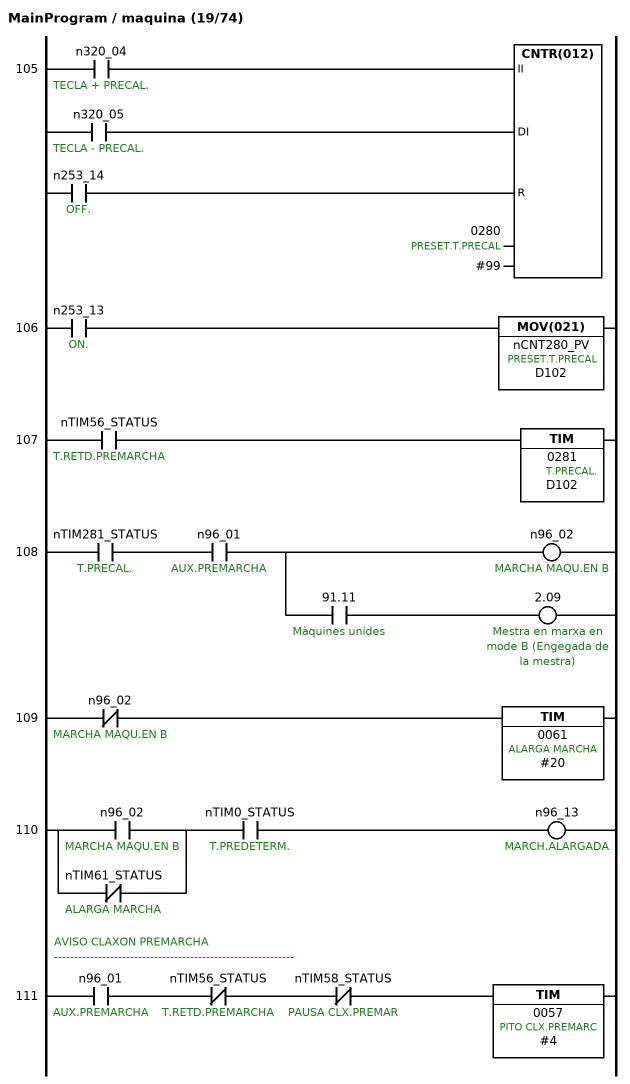
; [picture p24: MainProgram / maquina, rungs 105-111]
; rung 105
LD n320_04  ; TECLA + PRECAL.
LD n320_05  ; TECLA - PRECAL.
LD n253_14  ; OFF.
CNTR(012) 0280 #99  ; PRESET.T.PRECAL
; rung 106
LD n253_13  ; ON.
MOV(021) nCNT280_PV D102  ; PRESET.T.PRECAL
; rung 107
LD nTIM56_STATUS  ; T.RETD.PREMARCHA
TIM 0281 D102  ; T.PRECAL.
; rung 108
LD nTIM281_STATUS  ; T.PRECAL.
AND n96_01  ; AUX.PREMARCHA
OUT n96_02  ; MARCHA MAQU.EN B
AND 91.11  ; Màquines unides
OUT 2.09  ; Mestra en marxa en mode B (Engegada de la mestra)
; rung 109
LDNOT n96_02  ; MARCHA MAQU.EN B
TIM 0061 #20  ; ALARGA MARCHA
; rung 110
LD n96_02  ; MARCHA MAQU.EN B
ORNOT nTIM61_STATUS  ; ALARGA MARCHA
AND nTIM0_STATUS  ; T.PREDETERM.
OUT n96_13  ; MARCH.ALARGADA
; rung 111: AVISO CLAXON PREMARCHA / ------------------------------------------------------------
LD n96_01  ; AUX.PREMARCHA
ANDNOT nTIM56_STATUS  ; T.RETD.PREMARCHA
ANDNOT nTIM58_STATUS  ; PAUSA CLX.PREMAR
TIM 0057 #4  ; PITO CLX.PREMARC

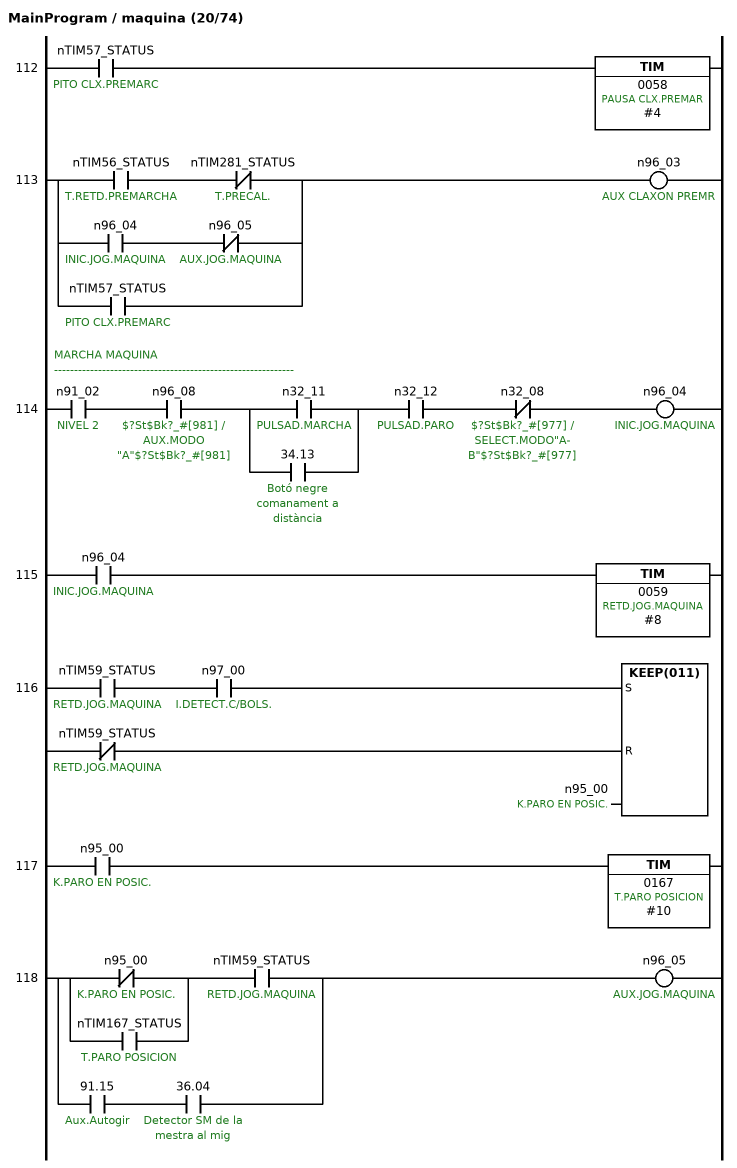
; rung 112
LD nTIM57_STATUS  ; PITO CLX.PREMARC
TIM 0058 #4  ; PAUSA CLX.PREMAR
; rung 113
LD nTIM56_STATUS  ; T.RETD.PREMARCHA
ANDNOT nTIM281_STATUS  ; T.PRECAL.
LD n96_04  ; INIC.JOG.MAQUINA
ANDNOT n96_05  ; AUX.JOG.MAQUINA
ORLD
OR nTIM57_STATUS  ; PITO CLX.PREMARC
OUT n96_03  ; AUX CLAXON PREMR
; rung 114: MARCHA MAQUINA / ------------------------------------------------------------
LD n91_02  ; NIVEL 2
AND n96_08  ; $?St$Bk?_#[981] / AUX.MODO "A"$?St$Bk?_#[981]
LD n32_11  ; PULSAD.MARCHA
OR 34.13  ; Botó negre comanament a distància
ANDLD
AND n32_12  ; PULSAD.PARO
ANDNOT n32_08  ; $?St$Bk?_#[977] / SELECT.MODO"A-B"$?St$Bk?_#[977]
OUT n96_04  ; INIC.JOG.MAQUINA
; rung 115
LD n96_04  ; INIC.JOG.MAQUINA
TIM 0059 #8  ; RETD.JOG.MAQUINA
; rung 116
LD nTIM59_STATUS  ; RETD.JOG.MAQUINA
AND n97_00  ; I.DETECT.C/BOLS.
LDNOT nTIM59_STATUS  ; RETD.JOG.MAQUINA
KEEP(011) n95_00  ; K.PARO EN POSIC.
; rung 117
LD n95_00  ; K.PARO EN POSIC.
TIM 0167 #10  ; T.PARO POSICION
; rung 118
LDNOT n95_00  ; K.PARO EN POSIC.
OR nTIM167_STATUS  ; T.PARO POSICION
AND nTIM59_STATUS  ; RETD.JOG.MAQUINA
LD 91.15  ; Aux.Autogir
AND 36.04  ; Detector SM de la mestra al mig
ORLD
OUT n96_05  ; AUX.JOG.MAQUINA

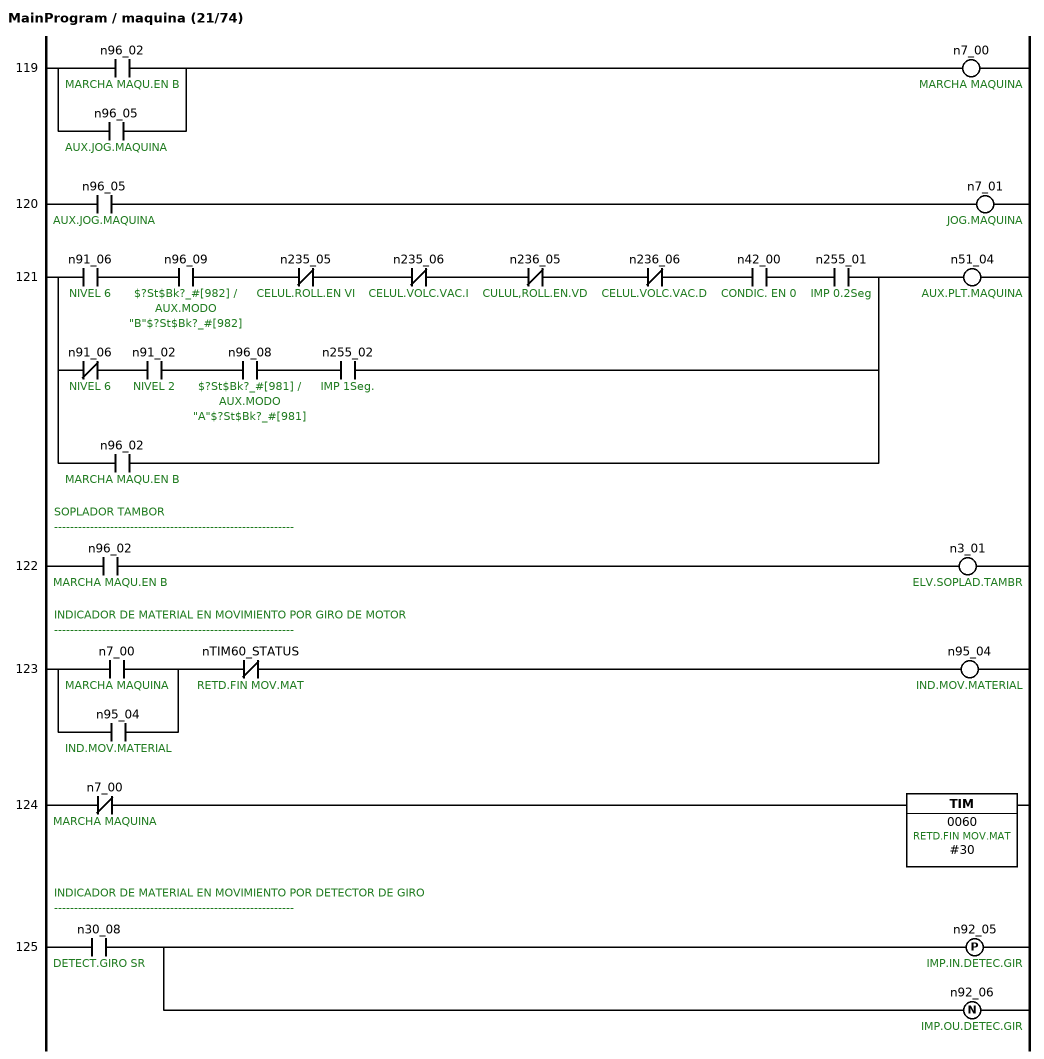
; rung 119
LD n96_02  ; MARCHA MAQU.EN B
OR n96_05  ; AUX.JOG.MAQUINA
OUT n7_00  ; MARCHA MAQUINA
; rung 120
LD n96_05  ; AUX.JOG.MAQUINA
OUT n7_01  ; JOG.MAQUINA
; rung 121
LD n91_06  ; NIVEL 6
AND n96_09  ; $?St$Bk?_#[982] / AUX.MODO "B"$?St$Bk?_#[982]
ANDNOT n235_05  ; CELUL.ROLL.EN VI
ANDNOT n235_06  ; CELUL.VOLC.VAC.I
ANDNOT n236_05  ; CULUL,ROLL.EN.VD
ANDNOT n236_06  ; CELUL.VOLC.VAC.D
AND n42_00  ; CONDIC. EN 0
AND n255_01  ; IMP 0.2Seg
LDNOT n91_06  ; NIVEL 6
AND n91_02  ; NIVEL 2
AND n96_08  ; $?St$Bk?_#[981] / AUX.MODO "A"$?St$Bk?_#[981]
AND n255_02  ; IMP 1Seg.
ORLD
OR n96_02  ; MARCHA MAQU.EN B
OUT n51_04  ; AUX.PLT.MAQUINA
; rung 122: SOPLADOR TAMBOR / ------------------------------------------------------------
LD n96_02  ; MARCHA MAQU.EN B
OUT n3_01  ; ELV.SOPLAD.TAMBR
; rung 123: INDICADOR DE MATERIAL EN MOVIMIENTO POR GIRO DE MOTOR / ------------------------------------------------------------
LD n7_00  ; MARCHA MAQUINA
OR n95_04  ; IND.MOV.MATERIAL
ANDNOT nTIM60_STATUS  ; RETD.FIN MOV.MAT
OUT n95_04  ; IND.MOV.MATERIAL
; rung 124
LDNOT n7_00  ; MARCHA MAQUINA
TIM 0060 #30  ; RETD.FIN MOV.MAT
; rung 125: INDICADOR DE MATERIAL EN MOVIMIENTO POR DETECTOR DE GIRO / ------------------------------------------------------------
LD n30_08  ; DETECT.GIRO SR
DIFU(013) n92_05  ; IMP.IN.DETEC.GIR
DIFD(014) n92_06  ; IMP.OU.DETEC.GIR  // IMPULSO DE SALIDA DETECT.DE GIRO

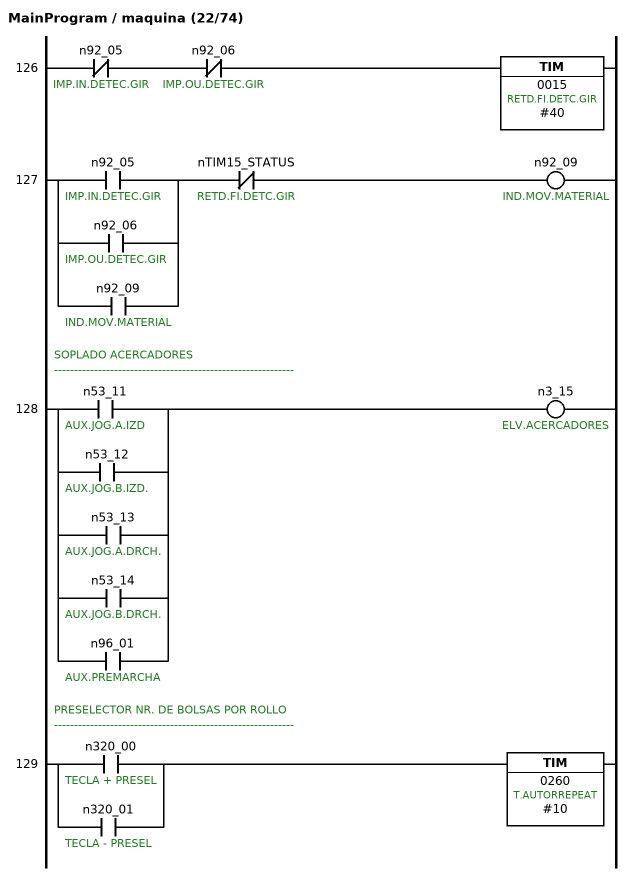
; rung 126
LDNOT n92_05  ; IMP.IN.DETEC.GIR
ANDNOT n92_06  ; IMP.OU.DETEC.GIR
TIM 0015 #40  ; RETD.FI.DETC.GIR  // T.RETARDO FIN DETECTOR DE GIRO
; rung 127
LD n92_05  ; IMP.IN.DETEC.GIR
OR n92_06  ; IMP.OU.DETEC.GIR
OR n92_09  ; IND.MOV.MATERIAL
ANDNOT nTIM15_STATUS  ; RETD.FI.DETC.GIR
OUT n92_09  ; IND.MOV.MATERIAL
; rung 128: SOPLADO ACERCADORES / ------------------------------------------------------------
LD n53_11  ; AUX.JOG.A.IZD
OR n53_12  ; AUX.JOG.B.IZD.
OR n53_13  ; AUX.JOG.A.DRCH.
OR n53_14  ; AUX.JOG.B.DRCH.
OR n96_01  ; AUX.PREMARCHA
OUT n3_15  ; ELV.ACERCADORES
; rung 129: PRESELECTOR NR. DE BOLSAS POR ROLLO / ------------------------------------------------------------
LD n320_00  ; TECLA + PRESEL
OR n320_01  ; TECLA - PRESEL
TIM 0260 #10  ; T.AUTORREPEAT

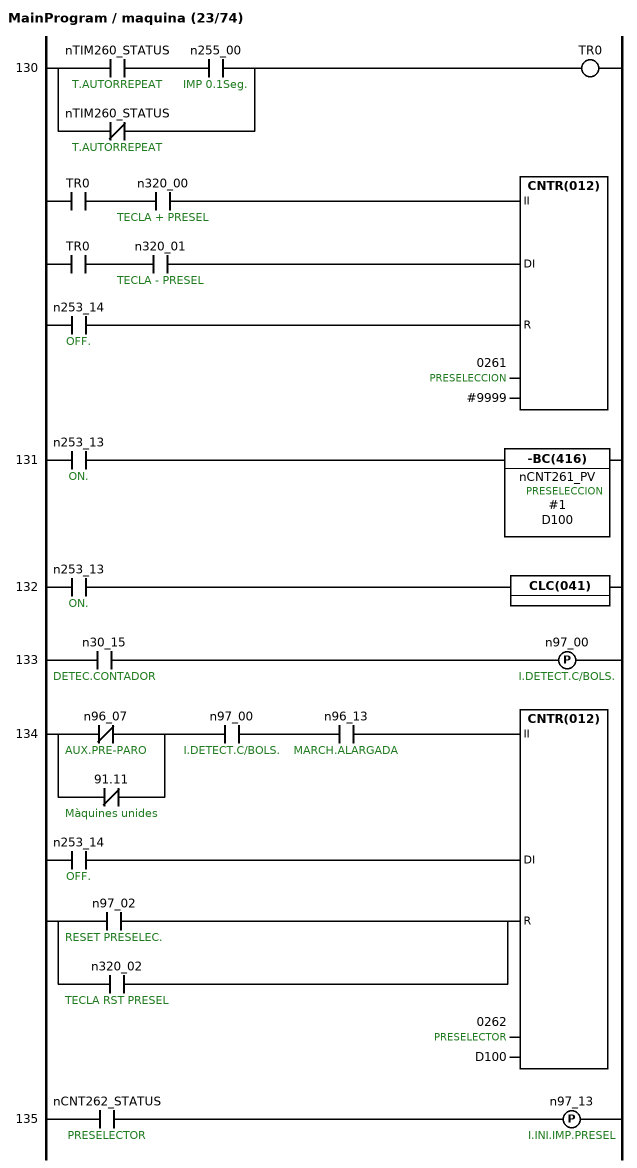
; rung 130
LD nTIM260_STATUS  ; T.AUTORREPEAT
AND n255_00  ; IMP 0.1Seg.
ORNOT nTIM260_STATUS  ; T.AUTORREPEAT
OUT TR0
AND n320_00  ; TECLA + PRESEL
LD TR0
AND n320_01  ; TECLA - PRESEL
LD n253_14  ; OFF.
CNTR(012) 0261 #9999  ; PRESELECCION
; rung 131
LD n253_13  ; ON.
-BC(416) nCNT261_PV #1 D100  ; PRESELECCION
; rung 132
LD n253_13  ; ON.
CLC(041)
; rung 133
LD n30_15  ; DETEC.CONTADOR
DIFU(013) n97_00  ; I.DETECT.C/BOLS.
; rung 134
LDNOT n96_07  ; AUX.PRE-PARO
ORNOT 91.11  ; Màquines unides
AND n97_00  ; I.DETECT.C/BOLS.
AND n96_13  ; MARCH.ALARGADA
LD n253_14  ; OFF.
LD n97_02  ; RESET PRESELEC.
OR n320_02  ; TECLA RST PRESEL
CNTR(012) 0262 D100  ; PRESELECTOR
; rung 135
LD nCNT262_STATUS  ; PRESELECTOR
DIFU(013) n97_13  ; I.INI.IMP.PRESEL

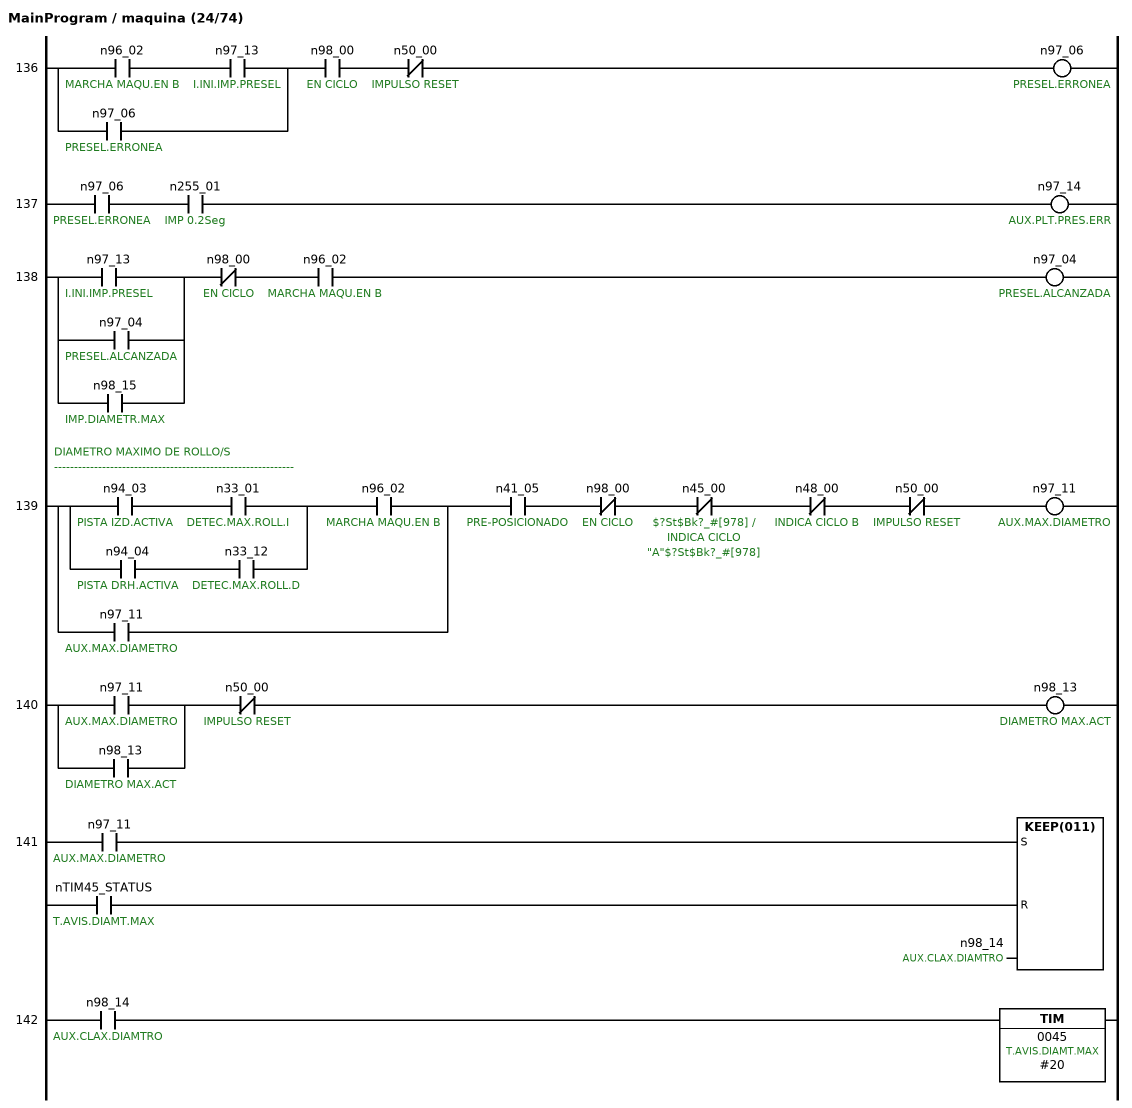
; rung 136
LD n96_02  ; MARCHA MAQU.EN B
AND n97_13  ; I.INI.IMP.PRESEL
OR n97_06  ; PRESEL.ERRONEA
AND n98_00  ; EN CICLO
ANDNOT n50_00  ; IMPULSO RESET
OUT n97_06  ; PRESEL.ERRONEA
; rung 137
LD n97_06  ; PRESEL.ERRONEA
AND n255_01  ; IMP 0.2Seg
OUT n97_14  ; AUX.PLT.PRES.ERR
; rung 138
LD n97_13  ; I.INI.IMP.PRESEL
OR n97_04  ; PRESEL.ALCANZADA
OR n98_15  ; IMP.DIAMETR.MAX
ANDNOT n98_00  ; EN CICLO
AND n96_02  ; MARCHA MAQU.EN B
OUT n97_04  ; PRESEL.ALCANZADA
; rung 139: DIAMETRO MAXIMO DE ROLLO/S / ------------------------------------------------------------
LD n94_03  ; PISTA IZD.ACTIVA
AND n33_01  ; DETEC.MAX.ROLL.I
LD n94_04  ; PISTA DRH.ACTIVA
AND n33_12  ; DETEC.MAX.ROLL.D
ORLD
AND n96_02  ; MARCHA MAQU.EN B
OR n97_11  ; AUX.MAX.DIAMETRO
AND n41_05  ; PRE-POSICIONADO
ANDNOT n98_00  ; EN CICLO
ANDNOT n45_00  ; $?St$Bk?_#[978] / INDICA CICLO "A"$?St$Bk?_#[978]
ANDNOT n48_00  ; INDICA CICLO B
ANDNOT n50_00  ; IMPULSO RESET
OUT n97_11  ; AUX.MAX.DIAMETRO
; rung 140
LD n97_11  ; AUX.MAX.DIAMETRO
OR n98_13  ; DIAMETRO MAX.ACT
ANDNOT n50_00  ; IMPULSO RESET
OUT n98_13  ; DIAMETRO MAX.ACT
; rung 141
LD n97_11  ; AUX.MAX.DIAMETRO
LD nTIM45_STATUS  ; T.AVIS.DIAMT.MAX
KEEP(011) n98_14  ; AUX.CLAX.DIAMTRO
; rung 142
LD n98_14  ; AUX.CLAX.DIAMTRO
TIM 0045 #20  ; T.AVIS.DIAMT.MAX

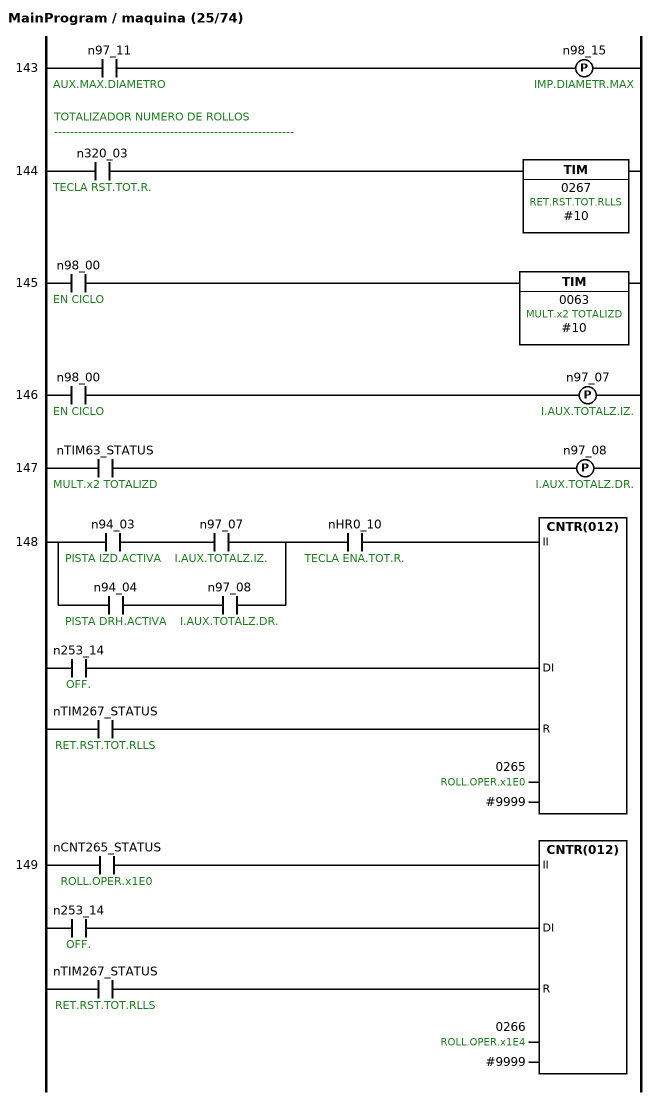
; rung 143
LD n97_11  ; AUX.MAX.DIAMETRO
DIFU(013) n98_15  ; IMP.DIAMETR.MAX
; rung 144: TOTALIZADOR NUMERO DE ROLLOS / ------------------------------------------------------------
LD n320_03  ; TECLA RST.TOT.R.
TIM 0267 #10  ; RET.RST.TOT.RLLS
; rung 145
LD n98_00  ; EN CICLO
TIM 0063 #10  ; MULT.x2 TOTALIZD
; rung 146
LD n98_00  ; EN CICLO
DIFU(013) n97_07  ; I.AUX.TOTALZ.IZ.
; rung 147
LD nTIM63_STATUS  ; MULT.x2 TOTALIZD
DIFU(013) n97_08  ; I.AUX.TOTALZ.DR.
; rung 148
LD n94_03  ; PISTA IZD.ACTIVA
AND n97_07  ; I.AUX.TOTALZ.IZ.
LD n94_04  ; PISTA DRH.ACTIVA
AND n97_08  ; I.AUX.TOTALZ.DR.
ORLD
AND nHR0_10  ; TECLA ENA.TOT.R.
LD n253_14  ; OFF.
LD nTIM267_STATUS  ; RET.RST.TOT.RLLS
CNTR(012) 0265 #9999  ; ROLL.OPER.x1E0
; rung 149
LD nCNT265_STATUS  ; ROLL.OPER.x1E0
LD n253_14  ; OFF.
LD nTIM267_STATUS  ; RET.RST.TOT.RLLS
CNTR(012) 0266 #9999  ; ROLL.OPER.x1E4

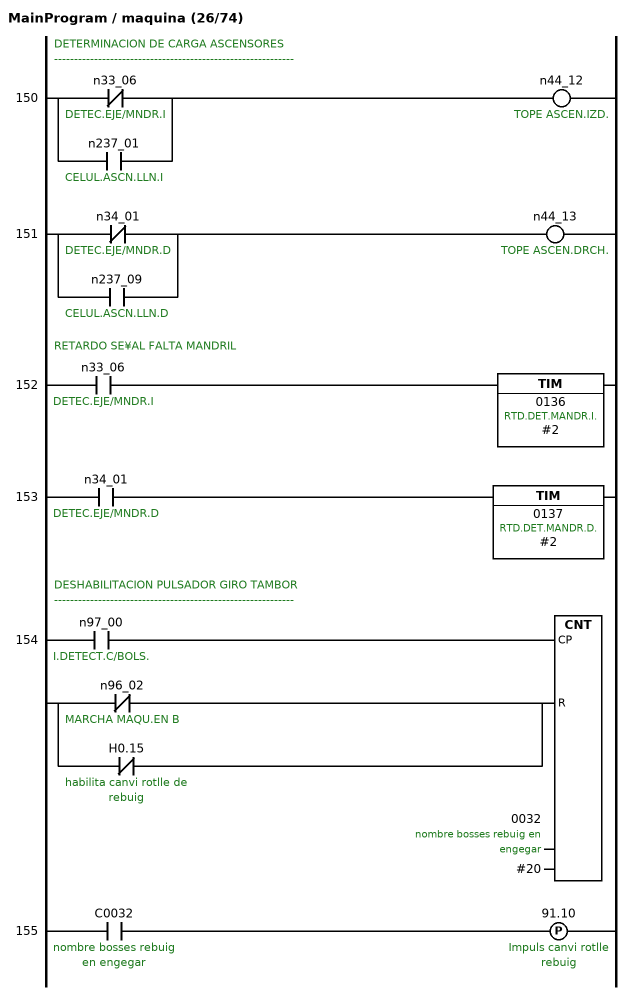
; rung 150: DETERMINACION DE CARGA ASCENSORES / ------------------------------------------------------------
LDNOT n33_06  ; DETEC.EJE/MNDR.I
OR n237_01  ; CELUL.ASCN.LLN.I
OUT n44_12  ; TOPE ASCEN.IZD.
; rung 151
LDNOT n34_01  ; DETEC.EJE/MNDR.D
OR n237_09  ; CELUL.ASCN.LLN.D
OUT n44_13  ; TOPE ASCEN.DRCH.
; rung 152: RETARDO SE¥AL FALTA MANDRIL
LD n33_06  ; DETEC.EJE/MNDR.I
TIM 0136 #2  ; RTD.DET.MANDR.I.
; rung 153
LD n34_01  ; DETEC.EJE/MNDR.D
TIM 0137 #2  ; RTD.DET.MANDR.D.
; rung 154: DESHABILITACION PULSADOR GIRO TAMBOR / ------------------------------------------------------------
LD n97_00  ; I.DETECT.C/BOLS.
LDNOT n96_02  ; MARCHA MAQU.EN B
ORNOT H0.15  ; habilita canvi rotlle de rebuig
CNT 0032 #20  ; nombre bosses rebuig en engegar
; rung 155
LD C0032  ; nombre bosses rebuig en engegar
DIFU(013) 91.10  ; Impuls canvi rotlle rebuig

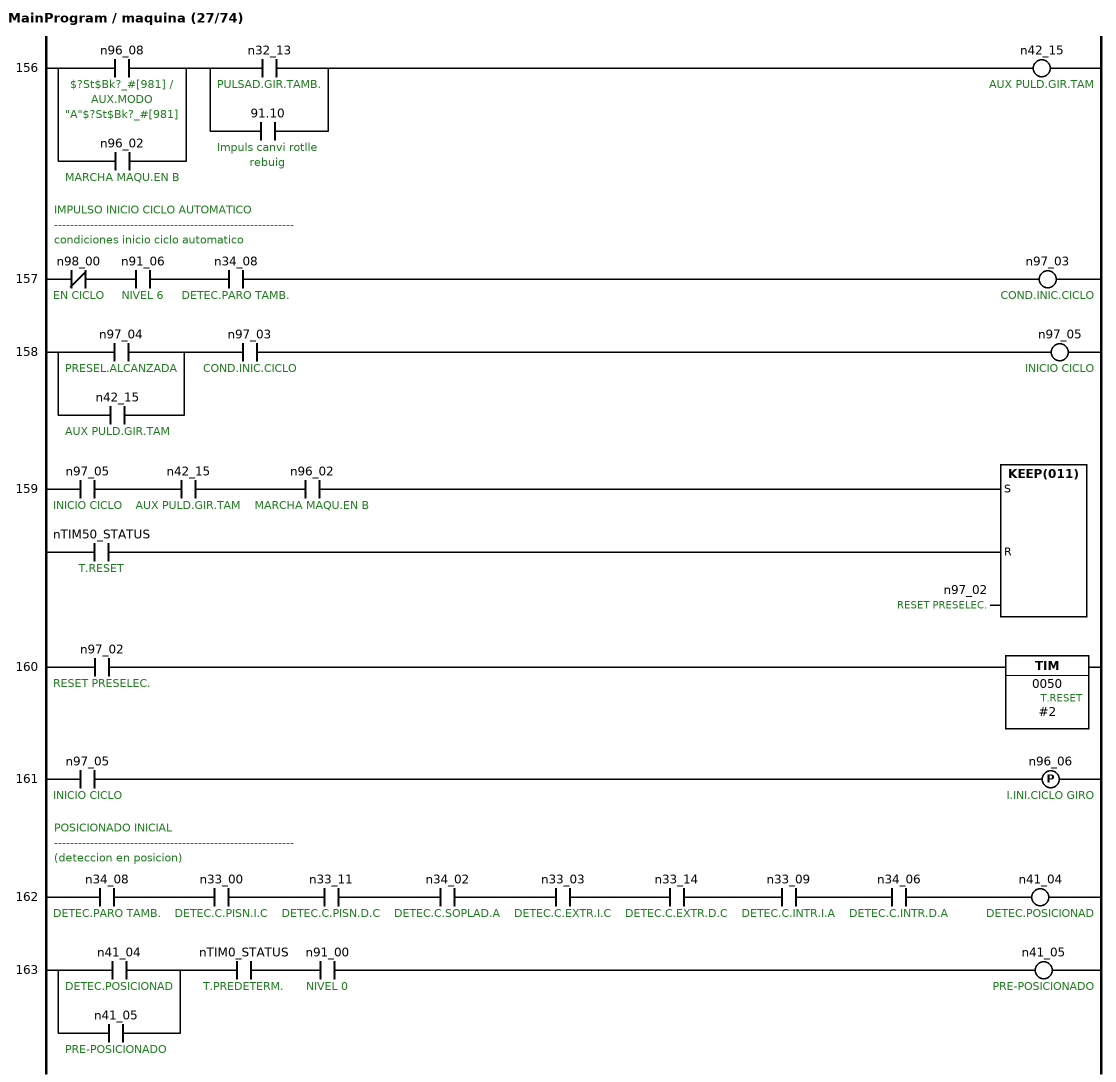
; rung 156
LD n96_08  ; $?St$Bk?_#[981] / AUX.MODO "A"$?St$Bk?_#[981]
OR n96_02  ; MARCHA MAQU.EN B
LD n32_13  ; PULSAD.GIR.TAMB.
OR 91.10  ; Impuls canvi rotlle rebuig
ANDLD
OUT n42_15  ; AUX PULD.GIR.TAM
; rung 157: IMPULSO INICIO CICLO AUTOMATICO / ------------------------------------------------------------ / condiciones inicio ciclo automatico
LDNOT n98_00  ; EN CICLO
AND n91_06  ; NIVEL 6
AND n34_08  ; DETEC.PARO TAMB.
OUT n97_03  ; COND.INIC.CICLO
; rung 158
LD n97_04  ; PRESEL.ALCANZADA
OR n42_15  ; AUX PULD.GIR.TAM
AND n97_03  ; COND.INIC.CICLO
OUT n97_05  ; INICIO CICLO
; rung 159
LD n97_05  ; INICIO CICLO
AND n42_15  ; AUX PULD.GIR.TAM
AND n96_02  ; MARCHA MAQU.EN B
LD nTIM50_STATUS  ; T.RESET
KEEP(011) n97_02  ; RESET PRESELEC.
; rung 160
LD n97_02  ; RESET PRESELEC.
TIM 0050 #2  ; T.RESET
; rung 161
LD n97_05  ; INICIO CICLO
DIFU(013) n96_06  ; I.INI.CICLO GIRO
; rung 162: POSICIONADO INICIAL / ------------------------------------------------------------ / (deteccion en posicion)
LD n34_08  ; DETEC.PARO TAMB.
AND n33_00  ; DETEC.C.PISN.I.C
AND n33_11  ; DETEC.C.PISN.D.C
AND n34_02  ; DETEC.C.SOPLAD.A
AND n33_03  ; DETEC.C.EXTR.I.C
AND n33_14  ; DETEC.C.EXTR.D.C
AND n33_09  ; DETEC.C.INTR.I.A
AND n34_06  ; DETEC.C.INTR.D.A
OUT n41_04  ; DETEC.POSICIONAD
; rung 163
LD n41_04  ; DETEC.POSICIONAD
OR n41_05  ; PRE-POSICIONADO
AND nTIM0_STATUS  ; T.PREDETERM.
AND n91_00  ; NIVEL 0
OUT n41_05  ; PRE-POSICIONADO

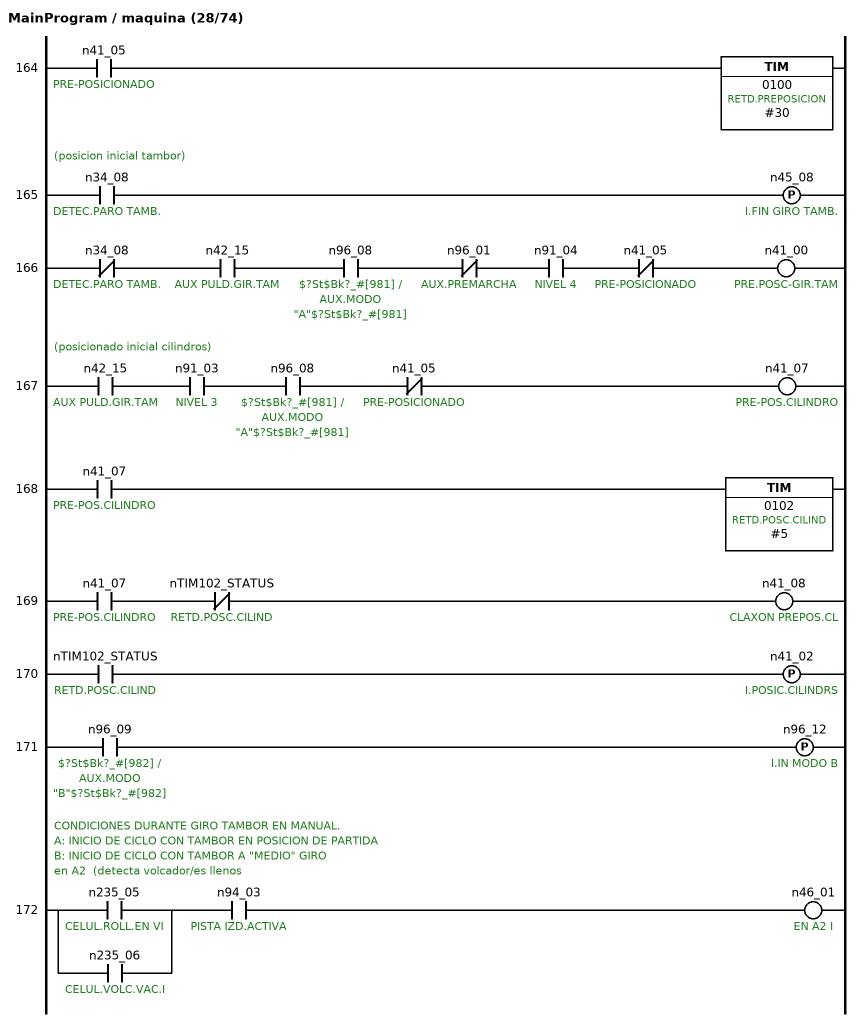
; rung 164
LD n41_05  ; PRE-POSICIONADO
TIM 0100 #30  ; RETD.PREPOSICION
; rung 165: (posicion inicial tambor)
LD n34_08  ; DETEC.PARO TAMB.
DIFU(013) n45_08  ; I.FIN GIRO TAMB.
; rung 166
LDNOT n34_08  ; DETEC.PARO TAMB.
AND n42_15  ; AUX PULD.GIR.TAM
AND n96_08  ; $?St$Bk?_#[981] / AUX.MODO "A"$?St$Bk?_#[981]
ANDNOT n96_01  ; AUX.PREMARCHA
AND n91_04  ; NIVEL 4
ANDNOT n41_05  ; PRE-POSICIONADO
OUT n41_00  ; PRE.POSC-GIR.TAM
; rung 167: (posicionado inicial cilindros)
LD n42_15  ; AUX PULD.GIR.TAM
AND n91_03  ; NIVEL 3
AND n96_08  ; $?St$Bk?_#[981] / AUX.MODO "A"$?St$Bk?_#[981]
ANDNOT n41_05  ; PRE-POSICIONADO
OUT n41_07  ; PRE-POS.CILINDRO
; rung 168
LD n41_07  ; PRE-POS.CILINDRO
TIM 0102 #5  ; RETD.POSC.CILIND
; rung 169
LD n41_07  ; PRE-POS.CILINDRO
ANDNOT nTIM102_STATUS  ; RETD.POSC.CILIND
OUT n41_08  ; CLAXON PREPOS.CL
; rung 170
LD nTIM102_STATUS  ; RETD.POSC.CILIND
DIFU(013) n41_02  ; I.POSIC.CILINDRS
; rung 171
LD n96_09  ; $?St$Bk?_#[982] / AUX.MODO "B"$?St$Bk?_#[982]
DIFU(013) n96_12  ; I.IN MODO B
; rung 172: CONDICIONES DURANTE GIRO TAMBOR EN MANUAL. / A: INICIO DE CICLO CON TAMBOR EN POSICION DE PARTIDA / B: INICIO DE CICLO CON TAMBOR A "MEDIO" GIRO / en A2  (detecta volcador/es llenos
LD n235_05  ; CELUL.ROLL.EN VI
OR n235_06  ; CELUL.VOLC.VAC.I
AND n94_03  ; PISTA IZD.ACTIVA
OUT n46_01  ; EN A2 I

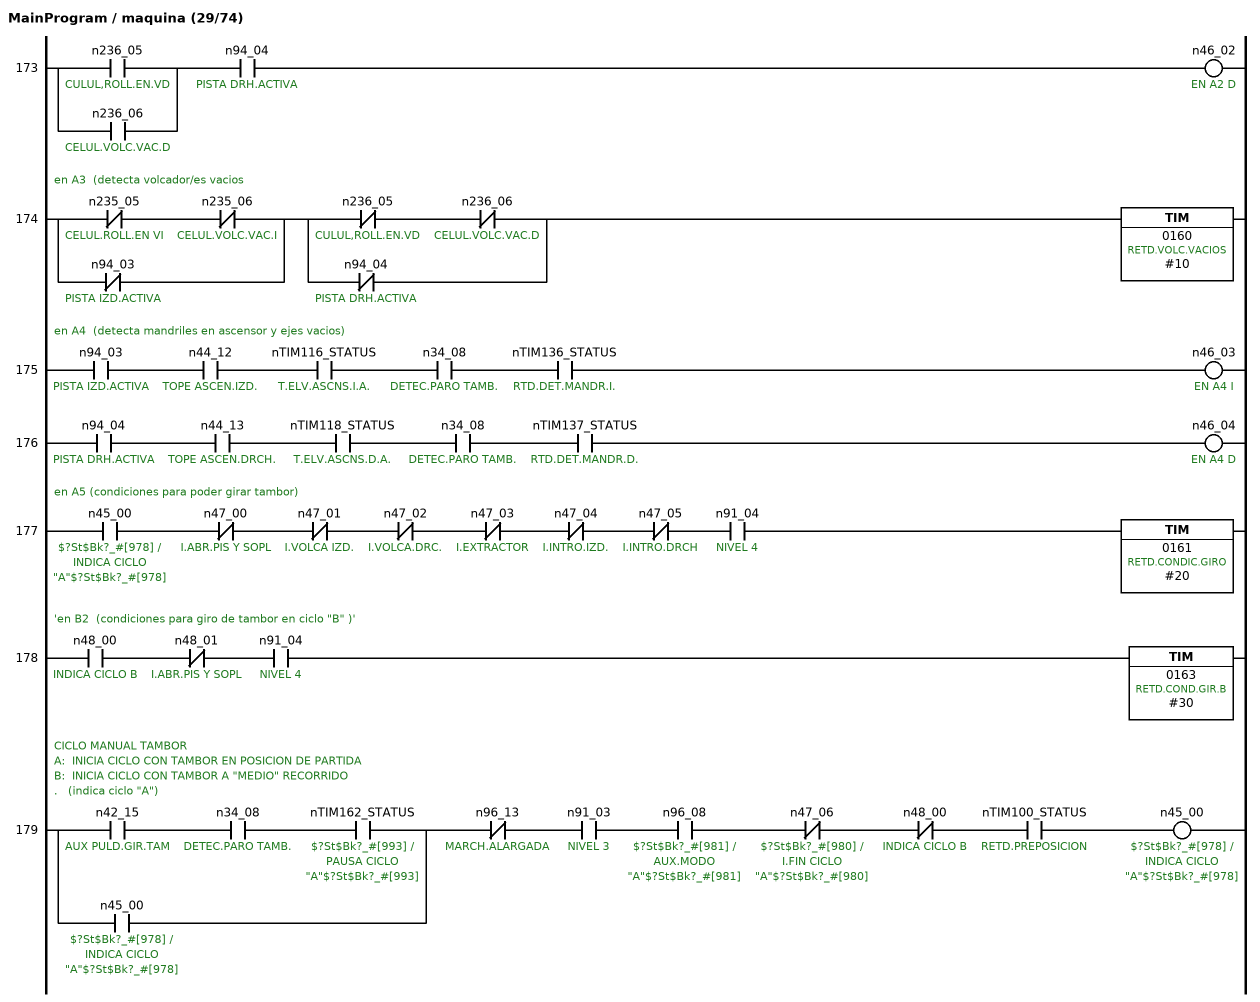
; rung 173
LD n236_05  ; CULUL,ROLL.EN.VD
OR n236_06  ; CELUL.VOLC.VAC.D
AND n94_04  ; PISTA DRH.ACTIVA
OUT n46_02  ; EN A2 D
; rung 174: en A3  (detecta volcador/es vacios
LDNOT n235_05  ; CELUL.ROLL.EN VI
ANDNOT n235_06  ; CELUL.VOLC.VAC.I
ORNOT n94_03  ; PISTA IZD.ACTIVA
LDNOT n236_05  ; CULUL,ROLL.EN.VD
ANDNOT n236_06  ; CELUL.VOLC.VAC.D
ORNOT n94_04  ; PISTA DRH.ACTIVA
ANDLD
TIM 0160 #10  ; RETD.VOLC.VACIOS
; rung 175: en A4  (detecta mandriles en ascensor y ejes vacios)
LD n94_03  ; PISTA IZD.ACTIVA
AND n44_12  ; TOPE ASCEN.IZD.
AND nTIM116_STATUS  ; T.ELV.ASCNS.I.A.
AND n34_08  ; DETEC.PARO TAMB.
AND nTIM136_STATUS  ; RTD.DET.MANDR.I.
OUT n46_03  ; EN A4 I
; rung 176
LD n94_04  ; PISTA DRH.ACTIVA
AND n44_13  ; TOPE ASCEN.DRCH.
AND nTIM118_STATUS  ; T.ELV.ASCNS.D.A.
AND n34_08  ; DETEC.PARO TAMB.
AND nTIM137_STATUS  ; RTD.DET.MANDR.D.
OUT n46_04  ; EN A4 D
; rung 177: en A5 (condiciones para poder girar tambor)
LD n45_00  ; $?St$Bk?_#[978] / INDICA CICLO "A"$?St$Bk?_#[978]
ANDNOT n47_00  ; I.ABR.PIS Y SOPL
ANDNOT n47_01  ; I.VOLCA IZD.
ANDNOT n47_02  ; I.VOLCA.DRC.
ANDNOT n47_03  ; I.EXTRACTOR
ANDNOT n47_04  ; I.INTRO.IZD.
ANDNOT n47_05  ; I.INTRO.DRCH
AND n91_04  ; NIVEL 4
TIM 0161 #20  ; RETD.CONDIC.GIRO
; rung 178: 'en B2  (condiciones para giro de tambor en ciclo "B" )'
LD n48_00  ; INDICA CICLO B
ANDNOT n48_01  ; I.ABR.PIS Y SOPL
AND n91_04  ; NIVEL 4
TIM 0163 #30  ; RETD.COND.GIR.B
; rung 179: CICLO MANUAL TAMBOR / A:  INICIA CICLO CON TAMBOR EN POSICION DE PARTIDA / B:  INICIA CICLO CON TAMBOR A "MEDIO" RECORRIDO / .   (indica ciclo "A")
LD n42_15  ; AUX PULD.GIR.TAM
AND n34_08  ; DETEC.PARO TAMB.
AND nTIM162_STATUS  ; $?St$Bk?_#[993] / PAUSA CICLO "A"$?St$Bk?_#[993]
OR n45_00  ; $?St$Bk?_#[978] / INDICA CICLO "A"$?St$Bk?_#[978]
ANDNOT n96_13  ; MARCH.ALARGADA
AND n91_03  ; NIVEL 3
AND n96_08  ; $?St$Bk?_#[981] / AUX.MODO "A"$?St$Bk?_#[981]
ANDNOT n47_06  ; $?St$Bk?_#[980] / I.FIN CICLO "A"$?St$Bk?_#[980]
ANDNOT n48_00  ; INDICA CICLO B
AND nTIM100_STATUS  ; RETD.PREPOSICION
OUT n45_00  ; $?St$Bk?_#[978] / INDICA CICLO "A"$?St$Bk?_#[978]

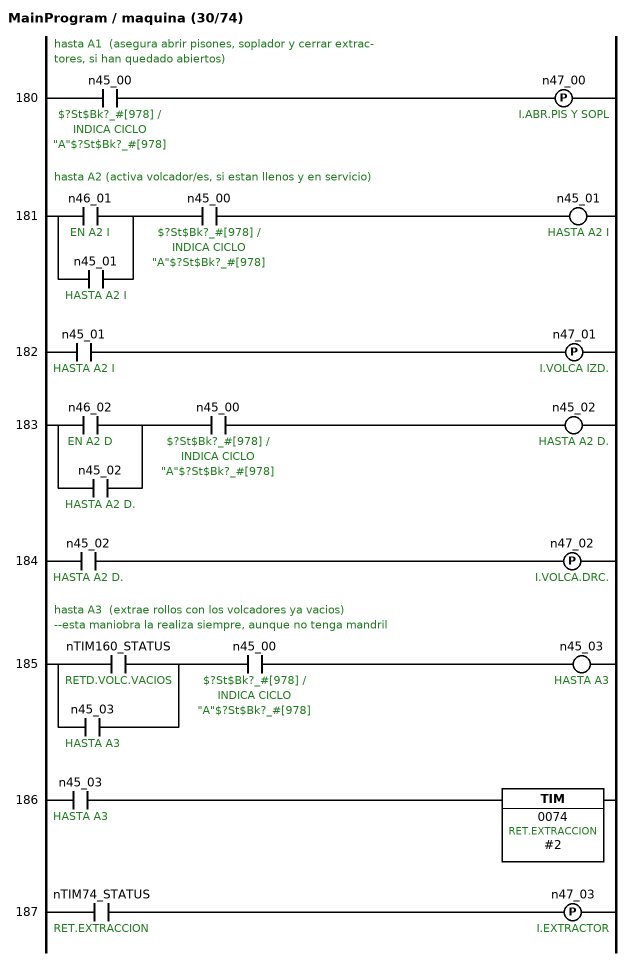
; rung 180: hasta A1  (asegura abrir pisones, soplador y cerrar extrac- / tores, si han quedado abiertos)
LD n45_00  ; $?St$Bk?_#[978] / INDICA CICLO "A"$?St$Bk?_#[978]
DIFU(013) n47_00  ; I.ABR.PIS Y SOPL
; rung 181: hasta A2 (activa volcador/es, si estan llenos y en servicio)
LD n46_01  ; EN A2 I
OR n45_01  ; HASTA A2 I
AND n45_00  ; $?St$Bk?_#[978] / INDICA CICLO "A"$?St$Bk?_#[978]
OUT n45_01  ; HASTA A2 I
; rung 182
LD n45_01  ; HASTA A2 I
DIFU(013) n47_01  ; I.VOLCA IZD.
; rung 183
LD n46_02  ; EN A2 D
OR n45_02  ; HASTA A2 D.
AND n45_00  ; $?St$Bk?_#[978] / INDICA CICLO "A"$?St$Bk?_#[978]
OUT n45_02  ; HASTA A2 D.
; rung 184
LD n45_02  ; HASTA A2 D.
DIFU(013) n47_02  ; I.VOLCA.DRC.
; rung 185: hasta A3  (extrae rollos con los volcadores ya vacios) / --esta maniobra la realiza siempre, aunque no tenga mandril
LD nTIM160_STATUS  ; RETD.VOLC.VACIOS
OR n45_03  ; HASTA A3
AND n45_00  ; $?St$Bk?_#[978] / INDICA CICLO "A"$?St$Bk?_#[978]
OUT n45_03  ; HASTA A3
; rung 186
LD n45_03  ; HASTA A3
TIM 0074 #2  ; RET.EXTRACCION
; rung 187
LD nTIM74_STATUS  ; RET.EXTRACCION
DIFU(013) n47_03  ; I.EXTRACTOR

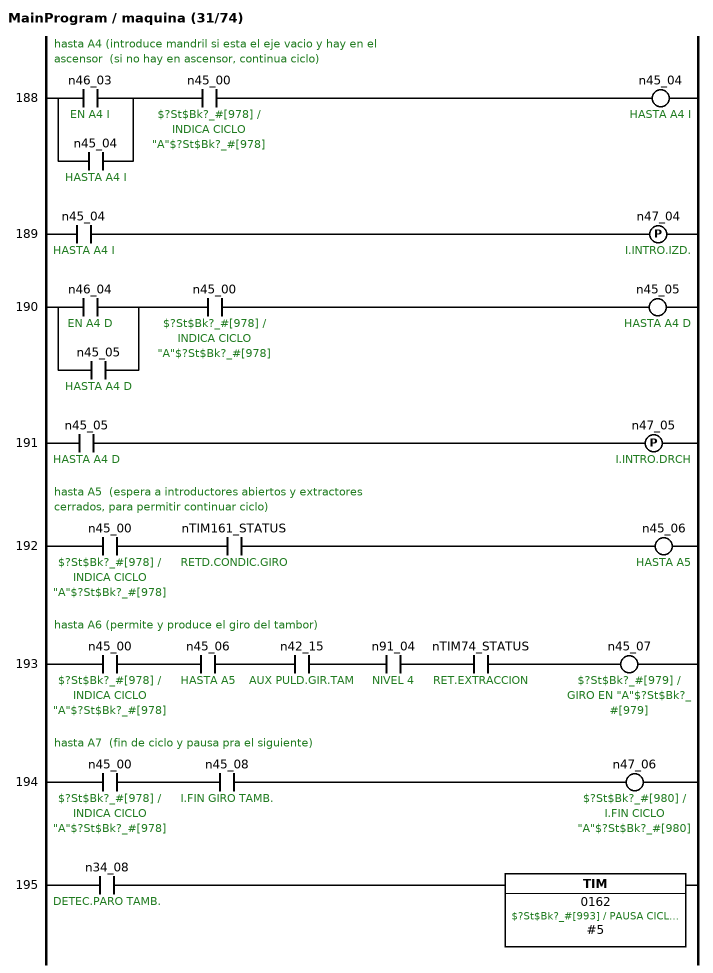
; rung 188: hasta A4 (introduce mandril si esta el eje vacio y hay en el / ascensor  (si no hay en ascensor, continua ciclo)
LD n46_03  ; EN A4 I
OR n45_04  ; HASTA A4 I
AND n45_00  ; $?St$Bk?_#[978] / INDICA CICLO "A"$?St$Bk?_#[978]
OUT n45_04  ; HASTA A4 I
; rung 189
LD n45_04  ; HASTA A4 I
DIFU(013) n47_04  ; I.INTRO.IZD.
; rung 190
LD n46_04  ; EN A4 D
OR n45_05  ; HASTA A4 D
AND n45_00  ; $?St$Bk?_#[978] / INDICA CICLO "A"$?St$Bk?_#[978]
OUT n45_05  ; HASTA A4 D
; rung 191
LD n45_05  ; HASTA A4 D
DIFU(013) n47_05  ; I.INTRO.DRCH
; rung 192: hasta A5  (espera a introductores abiertos y extractores / cerrados, para permitir continuar ciclo)
LD n45_00  ; $?St$Bk?_#[978] / INDICA CICLO "A"$?St$Bk?_#[978]
AND nTIM161_STATUS  ; RETD.CONDIC.GIRO
OUT n45_06  ; HASTA A5
; rung 193: hasta A6 (permite y produce el giro del tambor)
LD n45_00  ; $?St$Bk?_#[978] / INDICA CICLO "A"$?St$Bk?_#[978]
AND n45_06  ; HASTA A5
AND n42_15  ; AUX PULD.GIR.TAM
AND n91_04  ; NIVEL 4
AND nTIM74_STATUS  ; RET.EXTRACCION
OUT n45_07  ; $?St$Bk?_#[979] / GIRO EN "A"$?St$Bk?_#[979]
; rung 194: hasta A7  (fin de ciclo y pausa pra el siguiente)
LD n45_00  ; $?St$Bk?_#[978] / INDICA CICLO "A"$?St$Bk?_#[978]
AND n45_08  ; I.FIN GIRO TAMB.
OUT n47_06  ; $?St$Bk?_#[980] / I.FIN CICLO "A"$?St$Bk?_#[980]
; rung 195
LD n34_08  ; DETEC.PARO TAMB.
TIM 0162 #5  ; $?St$Bk?_#[993] / PAUSA CICLO "A"$?St$Bk?_#[993]

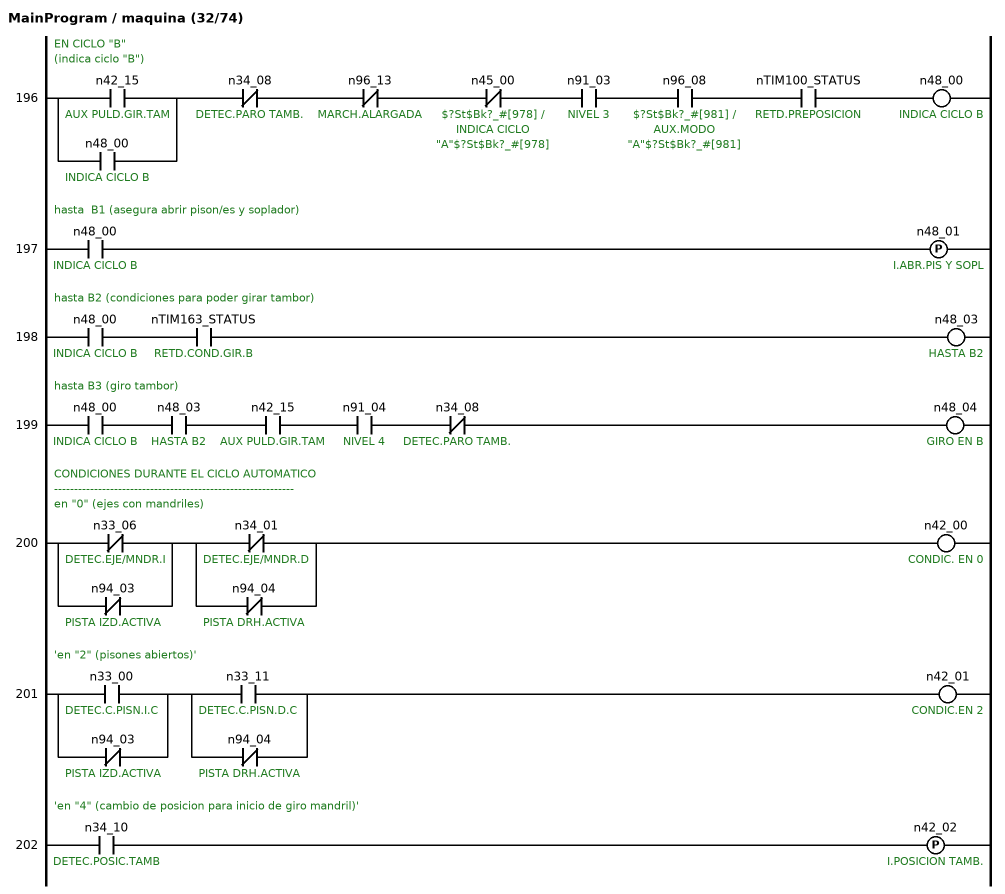
; rung 196: EN CICLO "B" / (indica ciclo "B")
LD n42_15  ; AUX PULD.GIR.TAM
OR n48_00  ; INDICA CICLO B
ANDNOT n34_08  ; DETEC.PARO TAMB.
ANDNOT n96_13  ; MARCH.ALARGADA
ANDNOT n45_00  ; $?St$Bk?_#[978] / INDICA CICLO "A"$?St$Bk?_#[978]
AND n91_03  ; NIVEL 3
AND n96_08  ; $?St$Bk?_#[981] / AUX.MODO "A"$?St$Bk?_#[981]
AND nTIM100_STATUS  ; RETD.PREPOSICION
OUT n48_00  ; INDICA CICLO B
; rung 197: hasta  B1 (asegura abrir pison/es y soplador)
LD n48_00  ; INDICA CICLO B
DIFU(013) n48_01  ; I.ABR.PIS Y SOPL
; rung 198: hasta B2 (condiciones para poder girar tambor)
LD n48_00  ; INDICA CICLO B
AND nTIM163_STATUS  ; RETD.COND.GIR.B
OUT n48_03  ; HASTA B2
; rung 199: hasta B3 (giro tambor)
LD n48_00  ; INDICA CICLO B
AND n48_03  ; HASTA B2
AND n42_15  ; AUX PULD.GIR.TAM
AND n91_04  ; NIVEL 4
ANDNOT n34_08  ; DETEC.PARO TAMB.
OUT n48_04  ; GIRO EN B
; rung 200: CONDICIONES DURANTE EL CICLO AUTOMATICO / ------------------------------------------------------------ / en "0" (ejes con mandriles)
LDNOT n33_06  ; DETEC.EJE/MNDR.I
ORNOT n94_03  ; PISTA IZD.ACTIVA
LDNOT n34_01  ; DETEC.EJE/MNDR.D
ORNOT n94_04  ; PISTA DRH.ACTIVA
ANDLD
OUT n42_00  ; CONDIC. EN 0
; rung 201: 'en "2" (pisones abiertos)'
LD n33_00  ; DETEC.C.PISN.I.C
ORNOT n94_03  ; PISTA IZD.ACTIVA
LD n33_11  ; DETEC.C.PISN.D.C
ORNOT n94_04  ; PISTA DRH.ACTIVA
ANDLD
OUT n42_01  ; CONDIC.EN 2
; rung 202: 'en "4" (cambio de posicion para inicio de giro mandril)'
LD n34_10  ; DETEC.POSIC.TAMB
DIFU(013) n42_02  ; I.POSICION TAMB.

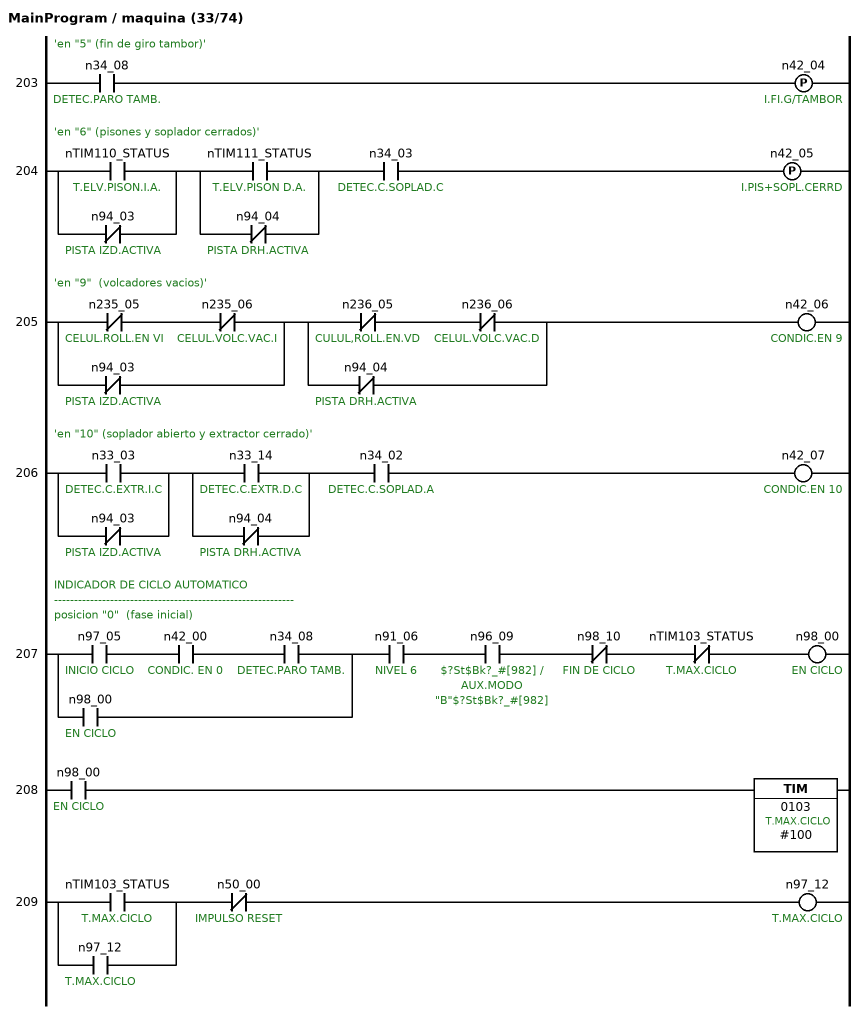
; rung 203: 'en "5" (fin de giro tambor)'
LD n34_08  ; DETEC.PARO TAMB.
DIFU(013) n42_04  ; I.FI.G/TAMBOR
; rung 204: 'en "6" (pisones y soplador cerrados)'
LD nTIM110_STATUS  ; T.ELV.PISON.I.A.
ORNOT n94_03  ; PISTA IZD.ACTIVA
LD nTIM111_STATUS  ; T.ELV.PISON D.A.
ORNOT n94_04  ; PISTA DRH.ACTIVA
ANDLD
AND n34_03  ; DETEC.C.SOPLAD.C
DIFU(013) n42_05  ; I.PIS+SOPL.CERRD
; rung 205: 'en "9"  (volcadores vacios)'
LDNOT n235_05  ; CELUL.ROLL.EN VI
ANDNOT n235_06  ; CELUL.VOLC.VAC.I
ORNOT n94_03  ; PISTA IZD.ACTIVA
LDNOT n236_05  ; CULUL,ROLL.EN.VD
ANDNOT n236_06  ; CELUL.VOLC.VAC.D
ORNOT n94_04  ; PISTA DRH.ACTIVA
ANDLD
OUT n42_06  ; CONDIC.EN 9
; rung 206: 'en "10" (soplador abierto y extractor cerrado)'
LD n33_03  ; DETEC.C.EXTR.I.C
ORNOT n94_03  ; PISTA IZD.ACTIVA
LD n33_14  ; DETEC.C.EXTR.D.C
ORNOT n94_04  ; PISTA DRH.ACTIVA
ANDLD
AND n34_02  ; DETEC.C.SOPLAD.A
OUT n42_07  ; CONDIC.EN 10
; rung 207: INDICADOR DE CICLO AUTOMATICO / ------------------------------------------------------------ / posicion "0"  (fase inicial)
LD n97_05  ; INICIO CICLO
AND n42_00  ; CONDIC. EN 0
AND n34_08  ; DETEC.PARO TAMB.
OR n98_00  ; EN CICLO
AND n91_06  ; NIVEL 6
AND n96_09  ; $?St$Bk?_#[982] / AUX.MODO "B"$?St$Bk?_#[982]
ANDNOT n98_10  ; FIN DE CICLO
ANDNOT nTIM103_STATUS  ; T.MAX.CICLO
OUT n98_00  ; EN CICLO
; rung 208
LD n98_00  ; EN CICLO
TIM 0103 #100  ; T.MAX.CICLO
; rung 209
LD nTIM103_STATUS  ; T.MAX.CICLO
OR n97_12  ; T.MAX.CICLO
ANDNOT n50_00  ; IMPULSO RESET
OUT n97_12  ; T.MAX.CICLO

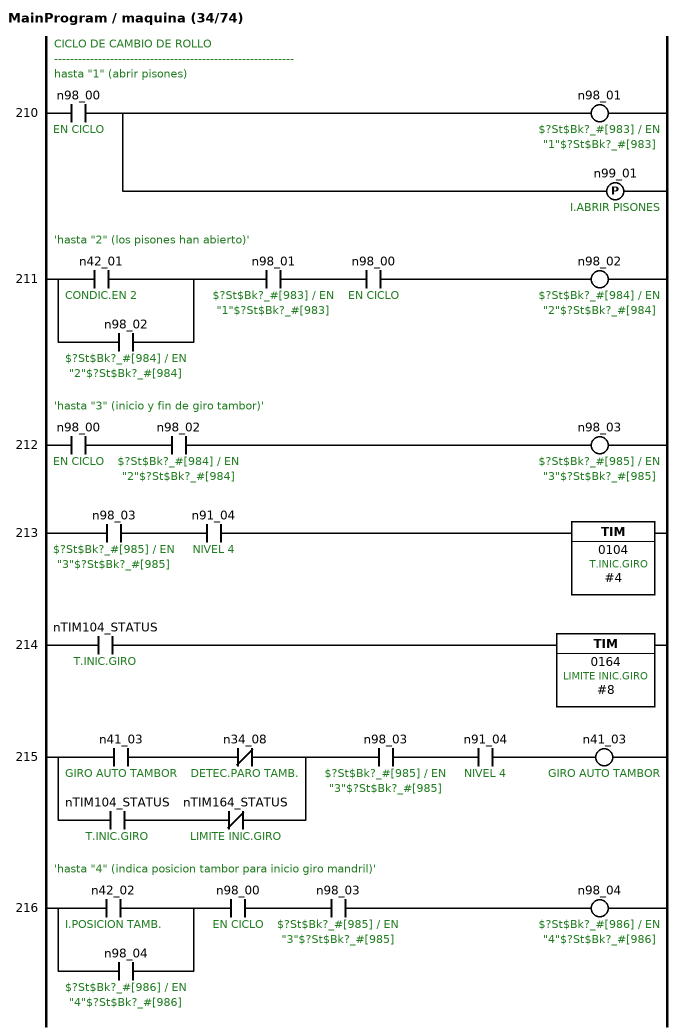
; rung 210: CICLO DE CAMBIO DE ROLLO / ------------------------------------------------------------ / hasta "1" (abrir pisones)
LD n98_00  ; EN CICLO
OUT n98_01  ; $?St$Bk?_#[983] / EN "1"$?St$Bk?_#[983]
DIFU(013) n99_01  ; I.ABRIR PISONES
; rung 211: 'hasta "2" (los pisones han abierto)'
LD n42_01  ; CONDIC.EN 2
OR n98_02  ; $?St$Bk?_#[984] / EN "2"$?St$Bk?_#[984]
AND n98_01  ; $?St$Bk?_#[983] / EN "1"$?St$Bk?_#[983]
AND n98_00  ; EN CICLO
OUT n98_02  ; $?St$Bk?_#[984] / EN "2"$?St$Bk?_#[984]
; rung 212: 'hasta "3" (inicio y fin de giro tambor)'
LD n98_00  ; EN CICLO
AND n98_02  ; $?St$Bk?_#[984] / EN "2"$?St$Bk?_#[984]
OUT n98_03  ; $?St$Bk?_#[985] / EN "3"$?St$Bk?_#[985]
; rung 213
LD n98_03  ; $?St$Bk?_#[985] / EN "3"$?St$Bk?_#[985]
AND n91_04  ; NIVEL 4
TIM 0104 #4  ; T.INIC.GIRO
; rung 214
LD nTIM104_STATUS  ; T.INIC.GIRO
TIM 0164 #8  ; LIMITE INIC.GIRO
; rung 215
LD n41_03  ; GIRO AUTO TAMBOR
ANDNOT n34_08  ; DETEC.PARO TAMB.
LD nTIM104_STATUS  ; T.INIC.GIRO
ANDNOT nTIM164_STATUS  ; LIMITE INIC.GIRO
ORLD
AND n98_03  ; $?St$Bk?_#[985] / EN "3"$?St$Bk?_#[985]
AND n91_04  ; NIVEL 4
OUT n41_03  ; GIRO AUTO TAMBOR
; rung 216: 'hasta "4" (indica posicion tambor para inicio giro mandril)'
LD n42_02  ; I.POSICION TAMB.
OR n98_04  ; $?St$Bk?_#[986] / EN "4"$?St$Bk?_#[986]
AND n98_00  ; EN CICLO
AND n98_03  ; $?St$Bk?_#[985] / EN "3"$?St$Bk?_#[985]
OUT n98_04  ; $?St$Bk?_#[986] / EN "4"$?St$Bk?_#[986]

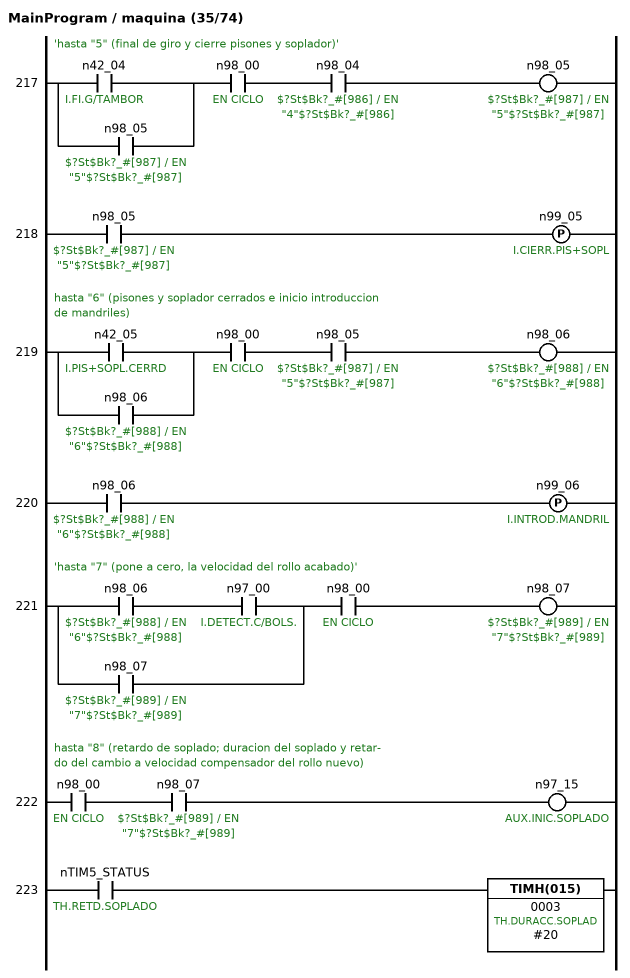
; rung 217: 'hasta "5" (final de giro y cierre pisones y soplador)'
LD n42_04  ; I.FI.G/TAMBOR
OR n98_05  ; $?St$Bk?_#[987] / EN "5"$?St$Bk?_#[987]
AND n98_00  ; EN CICLO
AND n98_04  ; $?St$Bk?_#[986] / EN "4"$?St$Bk?_#[986]
OUT n98_05  ; $?St$Bk?_#[987] / EN "5"$?St$Bk?_#[987]
; rung 218
LD n98_05  ; $?St$Bk?_#[987] / EN "5"$?St$Bk?_#[987]
DIFU(013) n99_05  ; I.CIERR.PIS+SOPL
; rung 219: hasta "6" (pisones y soplador cerrados e inicio introduccion / de mandriles)
LD n42_05  ; I.PIS+SOPL.CERRD
OR n98_06  ; $?St$Bk?_#[988] / EN "6"$?St$Bk?_#[988]
AND n98_00  ; EN CICLO
AND n98_05  ; $?St$Bk?_#[987] / EN "5"$?St$Bk?_#[987]
OUT n98_06  ; $?St$Bk?_#[988] / EN "6"$?St$Bk?_#[988]
; rung 220
LD n98_06  ; $?St$Bk?_#[988] / EN "6"$?St$Bk?_#[988]
DIFU(013) n99_06  ; I.INTROD.MANDRIL
; rung 221: 'hasta "7" (pone a cero, la velocidad del rollo acabado)'
LD n98_06  ; $?St$Bk?_#[988] / EN "6"$?St$Bk?_#[988]
AND n97_00  ; I.DETECT.C/BOLS.
OR n98_07  ; $?St$Bk?_#[989] / EN "7"$?St$Bk?_#[989]
AND n98_00  ; EN CICLO
OUT n98_07  ; $?St$Bk?_#[989] / EN "7"$?St$Bk?_#[989]
; rung 222: hasta "8" (retardo de soplado; duracion del soplado y retar- / do del cambio a velocidad compensador del rollo nuevo)
LD n98_00  ; EN CICLO
AND n98_07  ; $?St$Bk?_#[989] / EN "7"$?St$Bk?_#[989]
OUT n97_15  ; AUX.INIC.SOPLADO
; rung 223
LD nTIM5_STATUS  ; TH.RETD.SOPLADO
TIMH(015) 0003 #20  ; TH.DURACC.SOPLAD

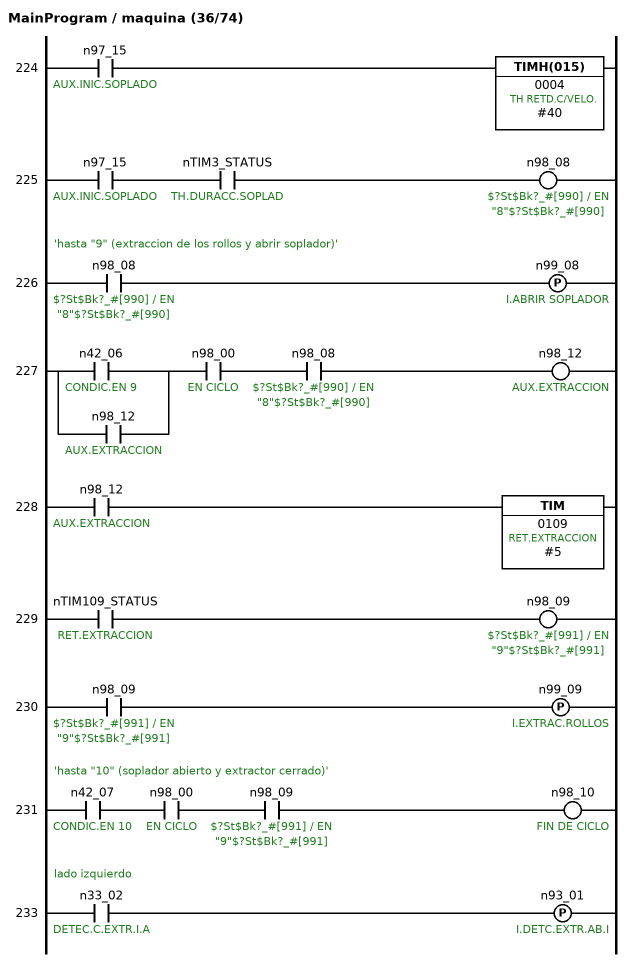
; rung 224
LD n97_15  ; AUX.INIC.SOPLADO
TIMH(015) 0004 #40  ; TH RETD.C/VELO.
; rung 225
LD n97_15  ; AUX.INIC.SOPLADO
AND nTIM3_STATUS  ; TH.DURACC.SOPLAD
OUT n98_08  ; $?St$Bk?_#[990] / EN "8"$?St$Bk?_#[990]
; rung 226: 'hasta "9" (extraccion de los rollos y abrir soplador)'
LD n98_08  ; $?St$Bk?_#[990] / EN "8"$?St$Bk?_#[990]
DIFU(013) n99_08  ; I.ABRIR SOPLADOR
; rung 227
LD n42_06  ; CONDIC.EN 9
OR n98_12  ; AUX.EXTRACCION
AND n98_00  ; EN CICLO
AND n98_08  ; $?St$Bk?_#[990] / EN "8"$?St$Bk?_#[990]
OUT n98_12  ; AUX.EXTRACCION
; rung 228
LD n98_12  ; AUX.EXTRACCION
TIM 0109 #5  ; RET.EXTRACCION
; rung 229
LD nTIM109_STATUS  ; RET.EXTRACCION
OUT n98_09  ; $?St$Bk?_#[991] / EN "9"$?St$Bk?_#[991]
; rung 230
LD n98_09  ; $?St$Bk?_#[991] / EN "9"$?St$Bk?_#[991]
DIFU(013) n99_09  ; I.EXTRAC.ROLLOS
; rung 231: 'hasta "10" (soplador abierto y extractor cerrado)'
LD n42_07  ; CONDIC.EN 10
AND n98_00  ; EN CICLO
AND n98_09  ; $?St$Bk?_#[991] / EN "9"$?St$Bk?_#[991]
OUT n98_10  ; FIN DE CICLO
; rung 232: VIGILANCIA ROLLOS NO CAIDOS DEL EJE REBOBINADOR / ------------------------------------------------------------
; rung 233: lado izquierdo
LD n33_02  ; DETEC.C.EXTR.I.A
DIFU(013) n93_01  ; I.DETC.EXTR.AB.I

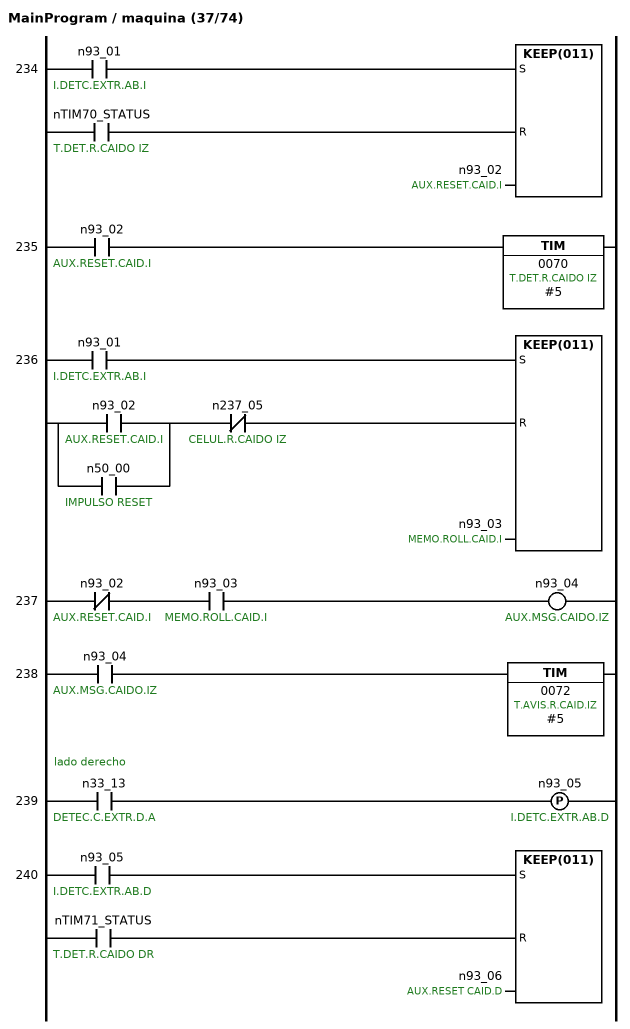
; rung 234
LD n93_01  ; I.DETC.EXTR.AB.I
LD nTIM70_STATUS  ; T.DET.R.CAIDO IZ
KEEP(011) n93_02  ; AUX.RESET.CAID.I
; rung 235
LD n93_02  ; AUX.RESET.CAID.I
TIM 0070 #5  ; T.DET.R.CAIDO IZ
; rung 236
LD n93_01  ; I.DETC.EXTR.AB.I
LD n93_02  ; AUX.RESET.CAID.I
OR n50_00  ; IMPULSO RESET
ANDNOT n237_05  ; CELUL.R.CAIDO IZ
KEEP(011) n93_03  ; MEMO.ROLL.CAID.I
; rung 237
LDNOT n93_02  ; AUX.RESET.CAID.I
AND n93_03  ; MEMO.ROLL.CAID.I
OUT n93_04  ; AUX.MSG.CAIDO.IZ
; rung 238
LD n93_04  ; AUX.MSG.CAIDO.IZ
TIM 0072 #5  ; T.AVIS.R.CAID.IZ
; rung 239: lado derecho
LD n33_13  ; DETEC.C.EXTR.D.A
DIFU(013) n93_05  ; I.DETC.EXTR.AB.D
; rung 240
LD n93_05  ; I.DETC.EXTR.AB.D
LD nTIM71_STATUS  ; T.DET.R.CAIDO DR
KEEP(011) n93_06  ; AUX.RESET CAID.D

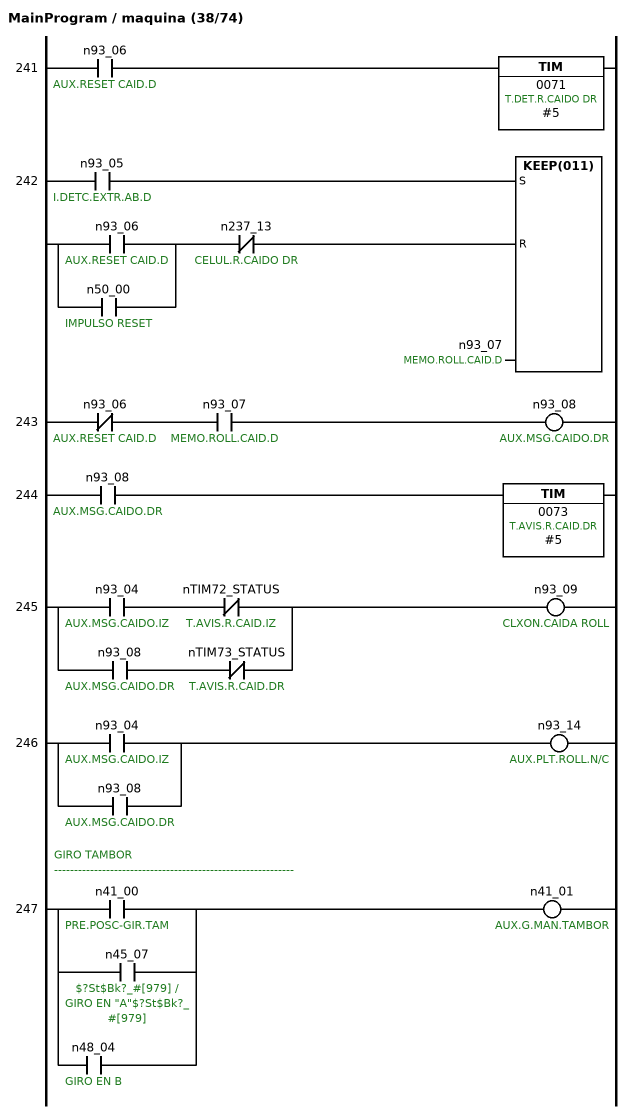
; rung 241
LD n93_06  ; AUX.RESET CAID.D
TIM 0071 #5  ; T.DET.R.CAIDO DR
; rung 242
LD n93_05  ; I.DETC.EXTR.AB.D
LD n93_06  ; AUX.RESET CAID.D
OR n50_00  ; IMPULSO RESET
ANDNOT n237_13  ; CELUL.R.CAIDO DR
KEEP(011) n93_07  ; MEMO.ROLL.CAID.D
; rung 243
LDNOT n93_06  ; AUX.RESET CAID.D
AND n93_07  ; MEMO.ROLL.CAID.D
OUT n93_08  ; AUX.MSG.CAIDO.DR
; rung 244
LD n93_08  ; AUX.MSG.CAIDO.DR
TIM 0073 #5  ; T.AVIS.R.CAID.DR
; rung 245
LD n93_04  ; AUX.MSG.CAIDO.IZ
ANDNOT nTIM72_STATUS  ; T.AVIS.R.CAID.IZ
LD n93_08  ; AUX.MSG.CAIDO.DR
ANDNOT nTIM73_STATUS  ; T.AVIS.R.CAID.DR
ORLD
OUT n93_09  ; CLXON.CAIDA ROLL
; rung 246
LD n93_04  ; AUX.MSG.CAIDO.IZ
OR n93_08  ; AUX.MSG.CAIDO.DR
OUT n93_14  ; AUX.PLT.ROLL.N/C
; rung 247: GIRO TAMBOR / ------------------------------------------------------------
LD n41_00  ; PRE.POSC-GIR.TAM
OR n45_07  ; $?St$Bk?_#[979] / GIRO EN "A"$?St$Bk?_#[979]
OR n48_04  ; GIRO EN B
OUT n41_01  ; AUX.G.MAN.TAMBOR

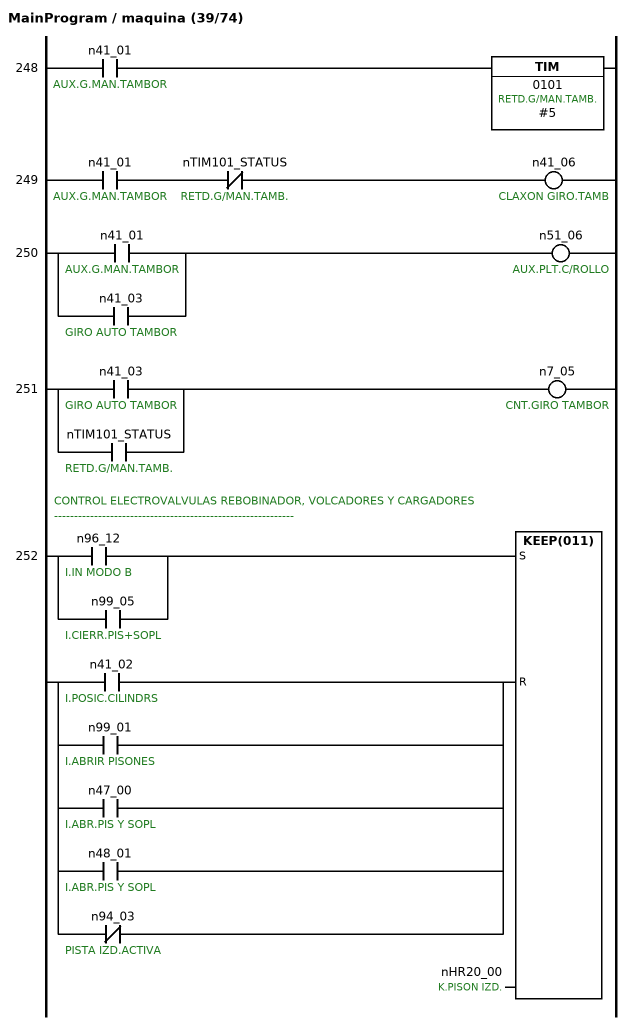
; rung 248
LD n41_01  ; AUX.G.MAN.TAMBOR
TIM 0101 #5  ; RETD.G/MAN.TAMB.
; rung 249
LD n41_01  ; AUX.G.MAN.TAMBOR
ANDNOT nTIM101_STATUS  ; RETD.G/MAN.TAMB.
OUT n41_06  ; CLAXON GIRO.TAMB
; rung 250
LD n41_01  ; AUX.G.MAN.TAMBOR
OR n41_03  ; GIRO AUTO TAMBOR
OUT n51_06  ; AUX.PLT.C/ROLLO
; rung 251
LD n41_03  ; GIRO AUTO TAMBOR
OR nTIM101_STATUS  ; RETD.G/MAN.TAMB.
OUT n7_05  ; CNT.GIRO TAMBOR
; rung 252: CONTROL ELECTROVALVULAS REBOBINADOR, VOLCADORES Y CARGADORES / ------------------------------------------------------------
LD n96_12  ; I.IN MODO B
OR n99_05  ; I.CIERR.PIS+SOPL
LD n41_02  ; I.POSIC.CILINDRS
OR n99_01  ; I.ABRIR PISONES
OR n47_00  ; I.ABR.PIS Y SOPL
OR n48_01  ; I.ABR.PIS Y SOPL
ORNOT n94_03  ; PISTA IZD.ACTIVA
KEEP(011) nHR20_00  ; K.PISON IZD.

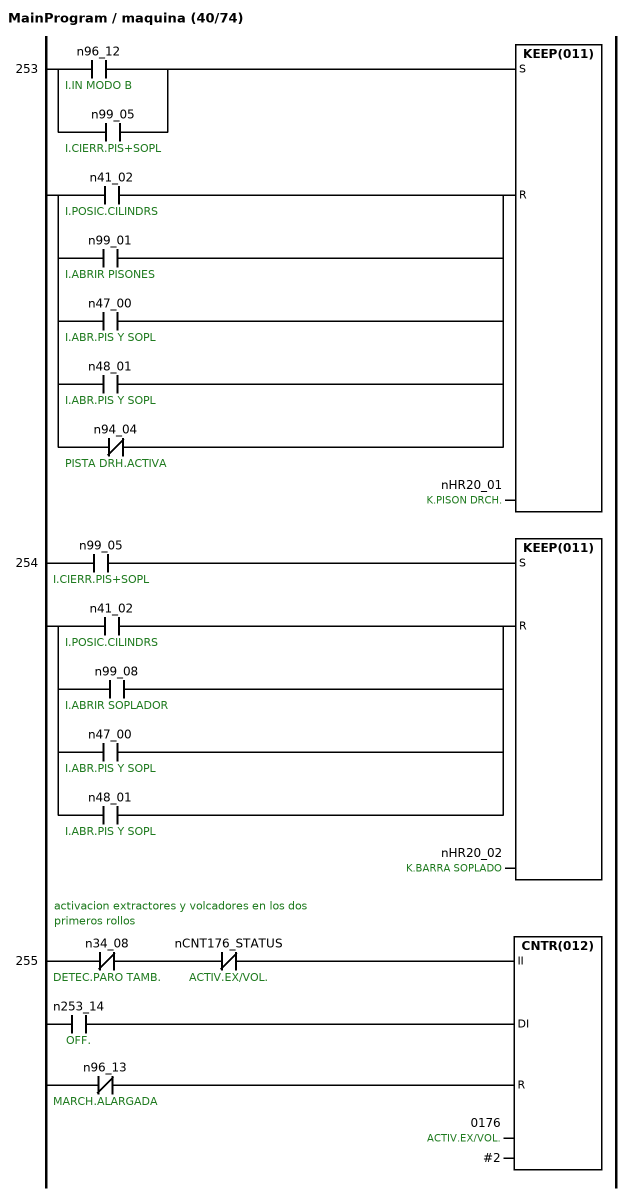
; rung 253
LD n96_12  ; I.IN MODO B
OR n99_05  ; I.CIERR.PIS+SOPL
LD n41_02  ; I.POSIC.CILINDRS
OR n99_01  ; I.ABRIR PISONES
OR n47_00  ; I.ABR.PIS Y SOPL
OR n48_01  ; I.ABR.PIS Y SOPL
ORNOT n94_04  ; PISTA DRH.ACTIVA
KEEP(011) nHR20_01  ; K.PISON DRCH.
; rung 254
LD n99_05  ; I.CIERR.PIS+SOPL
LD n41_02  ; I.POSIC.CILINDRS
OR n99_08  ; I.ABRIR SOPLADOR
OR n47_00  ; I.ABR.PIS Y SOPL
OR n48_01  ; I.ABR.PIS Y SOPL
KEEP(011) nHR20_02  ; K.BARRA SOPLADO
; rung 255: activacion extractores y volcadores en los dos / primeros rollos
LDNOT n34_08  ; DETEC.PARO TAMB.
ANDNOT nCNT176_STATUS  ; ACTIV.EX/VOL.
LD n253_14  ; OFF.
LDNOT n96_13  ; MARCH.ALARGADA
CNTR(012) 0176 #2  ; ACTIV.EX/VOL.

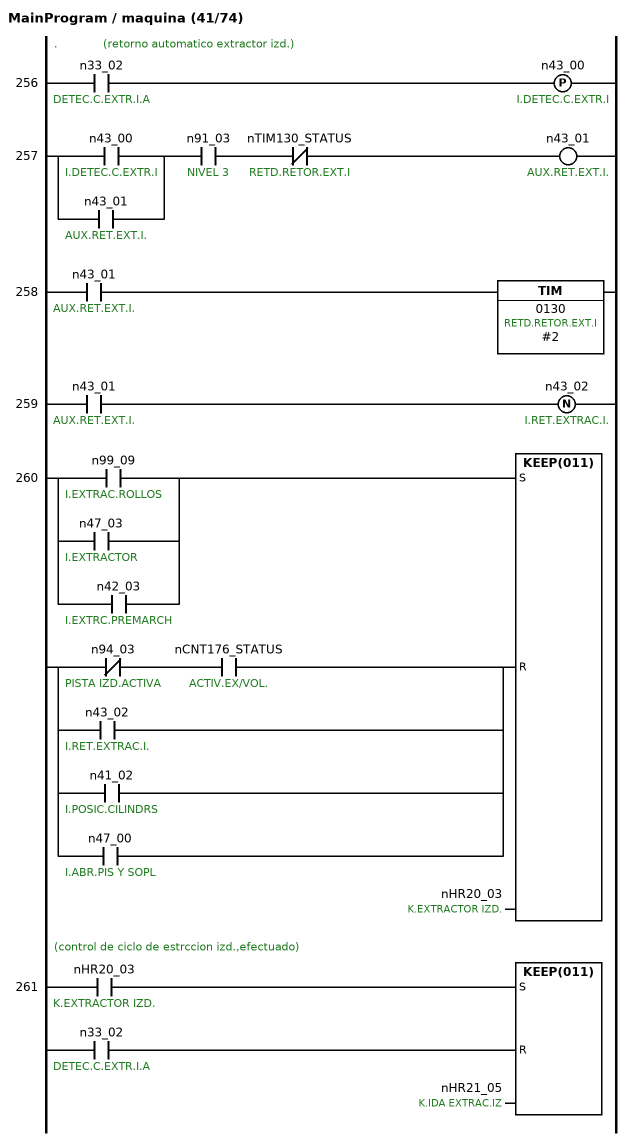
; rung 256: .             (retorno automatico extractor izd.)
LD n33_02  ; DETEC.C.EXTR.I.A
DIFU(013) n43_00  ; I.DETEC.C.EXTR.I
; rung 257
LD n43_00  ; I.DETEC.C.EXTR.I
OR n43_01  ; AUX.RET.EXT.I.
AND n91_03  ; NIVEL 3
ANDNOT nTIM130_STATUS  ; RETD.RETOR.EXT.I
OUT n43_01  ; AUX.RET.EXT.I.
; rung 258
LD n43_01  ; AUX.RET.EXT.I.
TIM 0130 #2  ; RETD.RETOR.EXT.I
; rung 259
LD n43_01  ; AUX.RET.EXT.I.
DIFD(014) n43_02  ; I.RET.EXTRAC.I.
; rung 260
LD n99_09  ; I.EXTRAC.ROLLOS
OR n47_03  ; I.EXTRACTOR
OR n42_03  ; I.EXTRC.PREMARCH
LDNOT n94_03  ; PISTA IZD.ACTIVA
AND nCNT176_STATUS  ; ACTIV.EX/VOL.
OR n43_02  ; I.RET.EXTRAC.I.
OR n41_02  ; I.POSIC.CILINDRS
OR n47_00  ; I.ABR.PIS Y SOPL
KEEP(011) nHR20_03  ; K.EXTRACTOR IZD.
; rung 261: (control de ciclo de estrccion izd.,efectuado)
LD nHR20_03  ; K.EXTRACTOR IZD.
LD n33_02  ; DETEC.C.EXTR.I.A
KEEP(011) nHR21_05  ; K.IDA EXTRAC.IZ

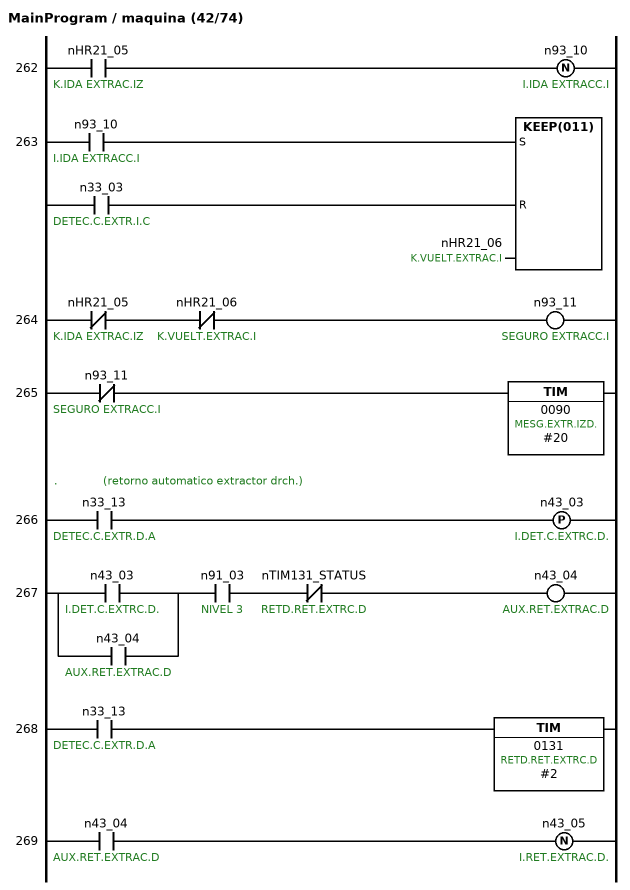
; rung 262
LD nHR21_05  ; K.IDA EXTRAC.IZ
DIFD(014) n93_10  ; I.IDA EXTRACC.I
; rung 263
LD n93_10  ; I.IDA EXTRACC.I
LD n33_03  ; DETEC.C.EXTR.I.C
KEEP(011) nHR21_06  ; K.VUELT.EXTRAC.I
; rung 264
LDNOT nHR21_05  ; K.IDA EXTRAC.IZ
ANDNOT nHR21_06  ; K.VUELT.EXTRAC.I
OUT n93_11  ; SEGURO EXTRACC.I
; rung 265
LDNOT n93_11  ; SEGURO EXTRACC.I
TIM 0090 #20  ; MESG.EXTR.IZD.
; rung 266: .             (retorno automatico extractor drch.)
LD n33_13  ; DETEC.C.EXTR.D.A
DIFU(013) n43_03  ; I.DET.C.EXTRC.D.
; rung 267
LD n43_03  ; I.DET.C.EXTRC.D.
OR n43_04  ; AUX.RET.EXTRAC.D
AND n91_03  ; NIVEL 3
ANDNOT nTIM131_STATUS  ; RETD.RET.EXTRC.D
OUT n43_04  ; AUX.RET.EXTRAC.D
; rung 268
LD n33_13  ; DETEC.C.EXTR.D.A
TIM 0131 #2  ; RETD.RET.EXTRC.D
; rung 269
LD n43_04  ; AUX.RET.EXTRAC.D
DIFD(014) n43_05  ; I.RET.EXTRAC.D.

